(* PLC project cam, Dassault Systèmes ControlBuild 2024x *)
(* stored: creationDateTime 2023-10-03T11:13:20-01:00 *)

(* This module simulates the behaviour of a cam (ovoid). *)
FUNCTION_BLOCK equipment_library.cam
  VAR_INPUT
    rotationSpeedRadS : REAL := 0.0;
    rotationSpeedDegS : REAL := 0.0;
  END_VAR
  VAR_OUTPUT
    positionTranslat : REAL := 0.0;
    percentTranslat : REAL := 0.0;
    incrementTranslat : REAL := 0.0;
  END_VAR
  VAR_OUTPUT
    angleRotationDeg : REAL := 0.0;
    angleRotationRad : REAL := 0.0;
  END_VAR
  VAR
    firstCycle : BOOL := false;
    incrementRotation : REAL := 0.0;
    oldPosition : REAL := 0.0;
  END_VAR
  VAR CONSTANT
    maxTranslat : REAL := 1000.0;
    initTranslat : REAL := 0.0;
    minTranslat : REAL := 0.0;
  END_VAR
  VAR
    d_locking : BOOL := false;
    v_d_locking : BOOL := false;
  END_VAR


ACTION C_source_code:
/* ----------------------------------------------------------------	*/
/* Type : Model of Operative Behaviour					*/
/* Category :  Actuators							*/
/* Author : Techniques Nouvelles d'Informatique				*/
/* Update date : October 2002						*/
/* ----------------------------------------------------------------	*/
/* This module simulate the behaviour of a cam (ovoid).		*/
/* The position of the cam goes from minTranslat to maxTranslat with	*/
/* the given rotation speed.						*/
/*										*/
/* nota : - the starting position is forced by initTranslat.		*/
/*	   - the speed setpoint can be set in				*/
/*		- radian per second	(rotationSpeedRadS)			*/
/*		- degree per second	(rotationSpeedDegS)			*/
/* ----------------------------------------------------------------	*/

/* Declaration of variables which don't need to be visualized during simulation */
float pi=3.1415926;


/* ----------------------------------------------------------------	*/
/* Initialization of the position of the cam for the first step of	*/
/* simulation.								*/
/* ----------------------------------------------------------------	*/
if (! firstCycle) {
	if (initTranslat > maxTranslat) positionTranslat = maxTranslat;
	else
		if (initTranslat < minTranslat) positionTranslat = minTranslat;
		else positionTranslat = initTranslat;

	firstCycle = 1;
	if ((maxTranslat - minTranslat) != 0.0)
		angleRotationRad = acos(1 - ((positionTranslat - minTranslat)/(maxTranslat - minTranslat)*2.0));
}

/* ----------------------------------------------------------------	*/
/* Rotation and translation (height of cam)				*/
/* ----------------------------------------------------------------	*/
if ((!d_locking) && ((rotationSpeedRadS!=0.0)||(rotationSpeedDegS!=0.0))) {

	/* compute the increment of rotation according to the clock of simulation	*/
	if (rotationSpeedRadS != 0.0) 
 		 incrementRotation= rotationSpeedRadS* (CLOCK_PERIOD/1000000.0) ;
	else
	if (rotationSpeedDegS != 0.0)
		incrementRotation= rotationSpeedDegS* 2*pi*(CLOCK_PERIOD/360000000.0) ;

	/* compute the angle of rotation (radian)	*/
	angleRotationRad = angleRotationRad + incrementRotation;
	if (angleRotationRad >= (2*pi)) {angleRotationRad -= 2*pi;}
	
	/* compute the position of translation	*/
	positionTranslat=(1 - cos(angleRotationRad))*(maxTranslat-minTranslat)/2.0 + minTranslat;
}

/* ----------------------------------------------------------------	*/
/* Compute the pecentage of height between the current position	*/
/* and the lowest and highest points of the cam				*/
/* ----------------------------------------------------------------	*/
percentTranslat = (100/(maxTranslat - minTranslat)) * (positionTranslat - minTranslat)  ;
		
/* ----------------------------------------------------------------	*/
/* Conversion of the rotation angle from radian to degree		*/
/* ----------------------------------------------------------------	*/
angleRotationDeg = (angleRotationRad*180)/pi;

/* ----------------------------------------------------------------	*/
/* Increment of translation							*/
/* ----------------------------------------------------------------	*/
incrementTranslat = positionTranslat - oldPosition;
oldPosition = positionTranslat;
END_ACTION

ACTION C_header:
#include <math.h>
END_ACTION
END_FUNCTION_BLOCK
